FUNCTION_BLOCK GrundstrukturSkill IMPLEMENTS I_State
VAR_INPUT
	bExecute			:BOOL;				// Trigger für Ausführung von Skill
	bReset				:BOOL;				// Trigger für Reset von Skill
	iObjState			:ObjectState;		// Information über Zustand von Objekt
	iSysState			:SystemState;		// Information über Zustand von System
END_VAR
VAR_OUTPUT
	iSkillCommand		:ObjectMode;		// Steuerungsvariable für Anlagenmodell
	bDone				:BOOL;				// Information ob Skill ausgfeührt wurde
	bBusy				:BOOL;				// Information ob Skill im Moment ausgeführt wird
	bLimit				:BOOL;				// Information ob Skill an einem Limit angekommen ist
	bError				:BOOL;				// Information ob sich Skill in Fehlerzustand befindet
	iErrorID			:INT;				// Information um welchen Fehler es sich handelt
END_VAR
VAR
	iState				:SkillState;		// Information über Zustand von Skill
	bTargetReached		:BOOL;				// Information ob Prozessziel erreicht wurde
	bLimitReached		:BOOL;				// Information ob Limit erreicht wurde
END_VAR

PROPERTY P_State : INT
GET
P_State := iState;
END_GET
END_PROPERTY

END_FUNCTION_BLOCK

(* stored: Version 1.1.0.1
   POU GrundstrukturSkill: Id {8849c73d-5d94-464c-8fa0-5cada18e040f}, SpecialFunc None
   Property P_State: Id {174b5214-bae6-4f3c-b2eb-b050fc2deeb8}
   Get Get: Id {611af6d0-4b12-4b33-98af-b90cc15ee0fa} *)
